// Checks if all elements in a boolean array are false.
FUNCTION F_AllAreFalse : BOOL // True if all elements in the array are false.
VAR_IN_OUT
	arValues : ARRAY[*] OF BOOL; // An array of boolean values to check.
END_VAR
VAR
	i : T_Position;
END_VAR

FOR i := LOWER_BOUND(arValues, 1) TO UPPER_BOUND(arValues, 1) DO
	IF arValues[i] THEN RETURN; END_IF 
	END_FOR
	
F_AllAreFalse := TRUE;

END_FUNCTION

(* stored: Version 1.1.0.1
   POU F_AllAreFalse: Id {84356fc4-7c14-0345-1147-2145684a68dc}, SpecialFunc None *)
